RoboDK station: Police_hand_UR5e.rdk

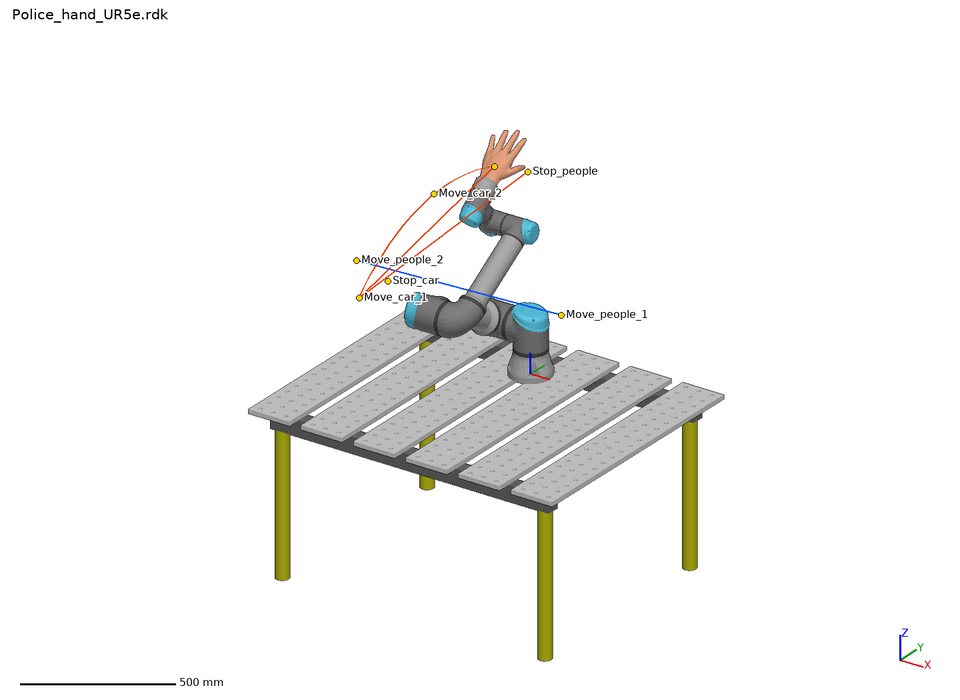
[picture v0: the station drawn from its stored meshes, robots at their saved joint values, targets as dots, program paths as lines]
Station Assistive_UR5e_SW (saved by RoboDK 5.9.2). Poses are relative to the parent item; angles as X-Y-Z fixed-axis rotations.
  - frame UR5e Base at (0, 0, 0) mm
    - robot UR5e: 6 axes, payload 5 kg, reach 850 mm, repeatability 0.03 mm, weight 18.4 kg
        modified DH rows (alpha deg, a mm, theta deg, d mm): 0, 0, 0, 162.5; 90, 0, 180, 0; 0, 425, 0, 0; 0, 392.25, 0, 133.3; -90, 0, 0, 99.7; 90, 0, 180, 99.6
        joint limits [-360, -360, -360, -360, -360, -360] to [360, 360, 360, 360, 360, 360]; home [0, -90, -90, 0, 90, 0]; saved at [-89.195, -155.935, 125.15, 166.621, -90.577, -90.561]
      - tool Hand, TCP at (0, 0, 50) mm, size 54.8 x 155.9 x 193.5 mm, geometry from Hand.stl
  - frame World at (0, 0, 0) mm
    - object Table at (0, 0, 0) mm, size 1193.8 x 965.2 x 609.6 mm, geometry from welding_table.sld
    - target Stop_car (Cartesian target) at (0, -800, 650) mm, rotated rx 0 ry 0 rz 90 deg; joints [-80.408, -173.15, 40.223, 222.927, -90, 80.408] of UR5e
    - target Move_people_1 (Cartesian target) at (420.93, -429.77, 500) mm, rotated rx 90 ry 0 rz 0 deg; joints [-18.362, -103.082, -73.522, -183.395, -18.362, 0] of UR5e
    - target Move_people_2 (Cartesian target) at (-348.29, -479.12, 500) mm, rotated rx 90 ry 0 rz 0 deg; joints [-120.445, -104.801, -101.385, -333.814, -239.555, 180] of UR5e
    - target Stop_people (joint target) at (200, -300, 900) mm; joints [101.992, 281.07, 53.116, 115.814, -90, -191.992] of UR5e
    - target Move_car_1 (Cartesian target) at (-131.59, -773.6, 543.02) mm, rotated rx 0 ry 37.75 rz -90 deg; joints [-89.856, 176.5, 66.408, 169.342, -89.912, -90.113] of UR5e
    - target Move_car_2 (Cartesian target) at (-131.59, -353.29, 748.73) mm, rotated rx 0 ry -4.59 rz -90 deg; joints [-89.732, 189.268, 103.877, 161.449, -90.021, -90.267] of UR5e
    - target Move_car_3 (Cartesian target) at (-131.59, -15.09, 712.31) mm, rotated rx 0 ry -45.84 rz -90 deg; joints [-89.195, 204.065, 125.15, 166.621, -90.577, -90.561] of UR5e
  - program Init (3 instructions, listed below)
  - program Priority_people (6 instructions, listed below)
  - program Priority_cars (7 instructions, listed below)
  - program MainProgram (3 instructions, listed below)
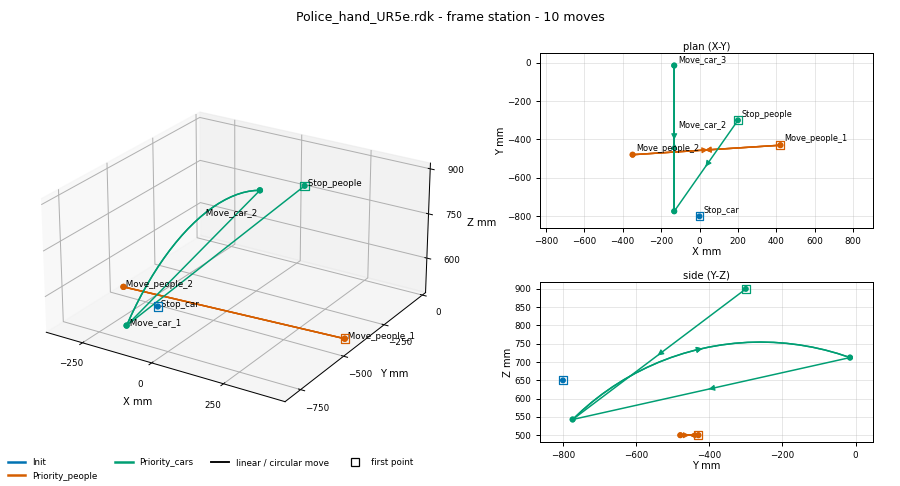
[picture p0: tool path of Police_hand_UR5e.rdk in frame station, 10 of 10 moves have a stored position in this frame; points joined in program order, loops and branches not executed]

--- program Init (robot UR5e) ---
  Est. Ref.: UR5e Base
  Est. herr: Hand
  MoveJ (Stop_car)

--- program Priority_people (robot UR5e) ---
  Est. Ref.: UR5e Base
  Est. herr: Hand
  MoveL (Move_people_1)
  MoveL (Move_people_2)
  MoveL (Move_people_1)
  MoveL (Move_people_2)

--- program Priority_cars (robot UR5e) ---
  Est. Ref.: UR5e Base
  Est. herr: Hand
  MoveL (Stop_people)
  MoveL (Move_car_1)
  MoveC (Move_car_2, Move_car_3)
  MoveL (Move_car_1)
  MoveC (Move_car_2, Move_car_3)

--- program MainProgram (robot UR5e) ---
  Llamar Init
  Llamar Priority_people
  Llamar Priority_cars
